TYPE (* ISOBUS UT split-bargraph object pool properties (two adjacent Linear Bar Graphs visualizing one signed value as two unsigned magnitude fills) *)
  (* Standard: 61499-2; Description: Copyright (c) 2026 Meisterschulen am Ostbahnhof This program and the accompanying materials are made available under the terms of the Eclipse Public License 2.0 which is available at https://www.eclipse.org/legal/epl-2.0/ SPDX-License-Identifier: EPL-2.0 *)
  (* Version 1.0, 2026-09-05, Franz Höpfinger, Meisterschulen am Ostbahnhof, initial API and implementation and/or initial documentation *)
  PACKAGE isobus::utils::bargraph;
  IMPORT logiBUS::utils::conversion::phys::NumericObjectPool_S;
  BargraphSplit_S : STRUCT
    stLeft : logiBUS::utils::conversion::phys::NumericObjectPool_S; (* Object pool properties of the Linear Bar Graph filling outward for negative values *)
    stRight : logiBUS::utils::conversion::phys::NumericObjectPool_S; (* Object pool properties of the Linear Bar Graph filling outward for positive values *)
    r32MinMagnitude : REAL := 0.0; (* Shared lower clamp bound for both sides' magnitude, matches both Bargraphs' own Min *)
    r32MaxMagnitude : REAL := 0.0; (* Shared upper clamp bound for both sides' magnitude, matches both Bargraphs' own Max *)
  END_STRUCT;
END_TYPE
